Universal Robots PolyScope program: ur3e_picking.urp

Program paulo_base_final (installation=paulo directory=/programs/usbdisk createdIn=3.2.19275.0 lastSavedIn=5.11.6.1010389 robotSerialNumber=20225300032)
Calibrated DH parameters: a=[-0.000184, -0.222113, -0.212499, 0.000052, -0.000121, 0]; d=[0.151687, 34.768241, -28.224416, -6.41321, 0.08539, 0.092028]; alpha=[1.5718, -0.002888, 0.002966, 1.571603, -1.571169, 0]; deltaTheta=[0, -0.424558, 0.515642, -0.091076, 0.000005, -0.000001]
InitVariablesNode variables(variable(name=ciclo, expression=0), variable(name=modo, expression=99), variable(name=pose_check, expression=0), variable(name=width, expression=0))
BeforeStart
  SafeHome (positionOptionType=SPEED_AND_ACCELERATION speed=1.047198 acceleration=1.396263 nextMotionTime=2)
  URCap 2FG Release (OnRobot, OnRobot A/S) dataModel(twofg.external-grip.target-width=0.0707000045776367, twofg.internal-grip.target-width=0.0847000045776367)
  Script: write_output_boolean_register(0, False )
  Wait Sleep waitTime=1
  Popup Message (haltProgram=false message=Ola, inicializar codigo e depois clicar ok. inputType=Text)
Robot Program (runOnlyOnce=false)
  Wait Sleep waitTime=1
  tmp := p[0,0,0,0,0,0]
  Script: write_output_integer_register(1,1)
  Script: sync()
  Wait Sleep waitTime=1
  Wait Condition expression=modo≠99 and pose_check≟0
  Folder Deteçao_Rotaçao [hidden by the author, left out]
  Folder Movimento [hidden by the author, left out]
  Script: write_output_integer_register(1,0)
  Script: write_output_integer_register(2,0)
  pose_check := 0
  Script: sync()
  SafeHome (positionOptionType=SPEED_AND_ACCELERATION speed=1.047198 acceleration=1.396263 nextMotionTime=2)
Thread Thread_2 (runOnlyOnce=false)
  Loop Forever
    modo := read_input_integer_register(0)
    ciclo := read_input_integer_register(1)
    width := read_input_float_register(6)
    pose_check := read_input_integer_register(2)
    Script: sync()
